PROGRAM PRG_1_PlcTask
VAR
END_VAR

PRG_2_PMPS_PRE();

// STUFF HERE

PRG_3_PMPS_POST();

END_PROGRAM

(* stored: Version 1.1.0.1, ProductVersion 3.1.4022.18
   POU PRG_1_PlcTask: Id {9c76104d-f8df-400f-b9a4-81d3480ca015}, SpecialFunc None *)
